TYPE SC_ACTUATOR_BeltConveyors :
(
	eBeltConveyorEntrance := 1,
	eBeltConveyorUpwards,
	eMaxNumBeltConveyors
)UINT;
END_TYPE

(* stored: Version 1.1.0.1, ProductVersion 3.1.4024.0
   DUT SC_ACTUATOR_BeltConveyors: Id {97b88d40-8bf1-4f6a-88d6-4b7718e5fb06} *)
